FUNCTION_BLOCK FB_Track IMPLEMENTS ITrack
VAR_INPUT
END_VAR
VAR_OUTPUT
END_VAR
VAR
	_list : ARRAY [1..iMaxNumbMovers] OF ST_MoverData;
	_sorted : ARRAY [1..iMaxNumbMovers] OF ST_MoverData;
	_sortedBU : ARRAY [1..iMaxNumbMovers] OF ST_MoverData;
	_tempData : ST_MoverData;
	_temp	: UDINT;
	_mover : ARRAY [1..10] OF IMover;
	i,j : INT;	
END_VAR

METHOD FindMover : UDINT
VAR_INPUT
	status	: INT;
END_VAR
FindMover := 0;
FOR i:= iMaxNumbMovers TO 1 BY -1 DO
	IF _sorted[i].status = status AND NOT _sorted[i].assigned THEN
		_sorted[i].assigned := TRUE;
		FindMover := _sorted[i].id;
		EXIT;
	END_IF
END_FOR
END_METHOD

METHOD SetMoverInUse : BOOL
VAR_INPUT
	moverNumber	: UDINT;
END_VAR
_Sorted[moverNumber].assigned := TRUE;
END_METHOD

METHOD SetMoverRef : BOOL
VAR_INPUT
	index	: DINT;
	mover	: IMover;
END_VAR
_mover[index]:= mover;
END_METHOD

METHOD Sort : BOOL
//backup Cycle Data
_sortedBU := _sorted;

// Step 1: Copy the list
_sorted := _list;

// Step 2: Restore Data
FOR i := 1 TO iMaxNumbMovers DO
	_sorted[i].assigned := _sortedBU[i].assigned;
END_FOR


// Step 2: Bubble Sort the list
FOR i := 1 TO iMaxNumbMovers - 1 DO
    FOR j := i + 1 TO iMaxNumbMovers DO
        IF _sorted[i].pos > _sorted[j].pos THEN
            _tempData := _sorted[i];
            _sorted[i] := _sorted[j];
            _sorted[j] := _tempData;
        END_IF
    END_FOR
END_FOR
END_METHOD

METHOD UpdateMoverData : BOOL
VAR_INPUT
	data	: ST_MoverData;
END_VAR
VAR
	temp	: INT;
END_VAR
_list[data.id] := data;
END_METHOD

END_FUNCTION_BLOCK

(* stored: Version 1.1.0.1, ProductVersion 3.1.4026.12
   POU FB_Track: Id {546a42d1-a9e5-46d3-b826-00988018d01d}, SpecialFunc None
   Method FindMover: Id {33981e48-82c3-4db8-b8e8-7ff5814bbbc3}
   Method SetMoverInUse: Id {87e123e5-04bd-4e13-99a7-1c2053f14a46}
   Method SetMoverRef: Id {bb3fa255-fee5-4b06-8ffa-9aff8162ff41}
   Method Sort: Id {5182b790-329f-48c5-abac-59d6da2e6290}
   Method UpdateMoverData: Id {19bcc54b-d09d-4767-9281-dabe045635c5} *)
